Omron Sysmac Studio project 17-408_20171120 (Sysmac Studio 1.19.0.13, StandardProject)

# Controller FS_17_408: NX1P2-9024DT version 1.13
Units and slaves: 節點1 : ASDA-A2-E CoE Drive (E001); 節點2 : ASDA-A2-E CoE Drive (E002)
Axis MC_Axis000, settings changed from default: AxisType=ServoType, FunctionLimit=SingleAxisPTP, UnitsConversion=EnumElement2, UnitsNumerator=1280000, UnitsDenominator=10, WorkGearRatio=16, MaxVelocity=500, MaxJogVelocity=500, HomingMode=BackupAndProximitySignalOn, HomingVelocity=10, HomingApproachVelocity=1, CompensationVelocity=1
Axis MC_Axis001, settings changed from default: AxisNumber=1, AxisType=ServoType, FunctionLimit=SingleAxisPTP, UnitsConversion=EnumElement2, UnitsNumerator=1280000, ReducerUse=EnumElement2, UnitsDenominator=11.75, TravelDistancePerWorkRotation=188, MotorGearRatio=16, MaxVelocity=600, MaxJogVelocity=600, HomingMode=BackupAndProximitySignalOn, HomingVelocity=20, HomingApproachVelocity=1, CompensationVelocity=1
Task PrimaryTask (priority 4, period or condition 2000): prAxis, prMainFlow, prSupplierNFeed, prInit, prError, prConverter

TYPE stAxis : STRUCT
    pbServoOn : BOOL;
    pbReset : BOOL;
    pbSerchHome : BOOL;
    pbJOGForward : BOOL;
    pbJOGBackward : BOOL;
    pbStop : BOOL;
    pbMoveAbs : BOOL;
    bMoveAbsDone : BOOL;
    bHoming : BOOL;
    bServoOn : BOOL;
    bAtPickPosition : BOOL;
    bAtLeavePickPosition : BOOL;
    bAtPutPosition : BOOL;
    bAtTHMoveSavePosition : BOOL;
    lrCurrentPosition : LREAL;
    lrMoveAbsAddData : LREAL;
    lrMoveAbsVelocity : LREAL;
    lrMoveJogVelocity : LREAL;
END_STRUCT END_TYPE

VAR_GLOBAL
    LS_THBack : BOOL;  (* 銅球節流回; at BuiltInIO://cpu/#0/Input_Bit_00; published *)
    LS_THOut : BOOL;  (* 銅球節流出; at BuiltInIO://cpu/#0/Input_Bit_01; published *)
    LS_MoveBack : BOOL;  (* 銅球前後回; at BuiltInIO://cpu/#0/Input_Bit_02; published *)
    LS_MoveOut : BOOL;  (* 銅球前後出; at BuiltInIO://cpu/#0/Input_Bit_03; published *)
    LS_ClipBack : BOOL;  (* 銅球夾持回; at BuiltInIO://cpu/#0/Input_Bit_04; published *)
    LS_ClipOut : BOOL;  (* 銅球夾持出; at BuiltInIO://cpu/#0/Input_Bit_05; published *)
    SNR_MCInPosition : BOOL;  (* 設備定位檢知; at BuiltInIO://cpu/#0/Input_Bit_08; published *)
    SNR_Feed : BOOL;  (* 銅球進料檢知; at BuiltInIO://cpu/#0/Input_Bit_09; published *)
    SNR_Full : BOOL;  (* 銅球滿料檢知; at BuiltInIO://cpu/#0/Input_Bit_10; published *)
    Ex_StartFlag : BOOL;  (* 外部設備送料起動; at BuiltInIO://cpu/#0/Input_Bit_12; published *)
    Ex_ClipOn : BOOL;  (* 外部設備已夾持; at BuiltInIO://cpu/#0/Input_Bit_13; published *)
    SOL_TH : BOOL;  (* 銅球節流電磁閥; at BuiltInIO://cpu/#0/Output_Bit_00; published *)
    SOL_Move : BOOL;  (* 銅球前後電磁閥; at BuiltInIO://cpu/#0/Output_Bit_01; published *)
    SOL_Clip : BOOL;  (* 銅球夾持電磁閥; at BuiltInIO://cpu/#0/Output_Bit_02; published *)
    SOL_FixBack : BOOL;  (* 定位氣壓夾爪回電磁閥; at BuiltInIO://cpu/#0/Output_Bit_03; published *)
    SOL_FixUpBack : BOOL;  (* 上振動定位氣壓夾爪回電磁閥; at BuiltInIO://cpu/#0/Output_Bit_04; published *)
    RY_Full : BOOL;  (* 振動筒繼電器; at BuiltInIO://cpu/#0/Output_Bit_05; published *)
    RY_Feed : BOOL;  (* 平送繼電器; at BuiltInIO://cpu/#0/Output_Bit_06; published *)
    RY_Brake : BOOL;  (* 上下軸剎車繼電器; at BuiltInIO://cpu/#0/Output_Bit_07; published *)
    Ex_FinishFlag : BOOL;  (* 外部設備送料完成; at BuiltInIO://cpu/#0/Output_Bit_08; published *)
    Ex_MachineReday : BOOL;  (* 外部設備可動作; at BuiltInIO://cpu/#0/Output_Bit_09; published *)
    SOL_FixOut : BOOL;  (* 定位氣壓夾爪出電磁閥; at IOBus://unit#2/Output Bit 16 bits/Output Bit 00; published *)
    SOL_FixUpOut : BOOL;  (* 上振動定位氣壓夾爪出電磁閥; at IOBus://unit#2/Output Bit 16 bits/Output Bit 02; published *)
    SOL_FixDownBack : BOOL;  (* 下振動定位氣壓夾爪回電磁閥; at IOBus://unit#2/Output Bit 16 bits/Output Bit 04; published *)
    SOL_FixDownOut : BOOL;  (* 下振動定位氣壓夾爪出電磁閥; at IOBus://unit#2/Output Bit 16 bits/Output Bit 06; published *)
    BZ : BOOL;  (* 蜂鳴器; at IOBus://unit#2/Output Bit 16 bits/Output Bit 01 *)
    YL : BOOL;  (* 黃燈; at IOBus://unit#2/Output Bit 16 bits/Output Bit 03 *)
    GL : BOOL;  (* 綠燈; at IOBus://unit#2/Output Bit 16 bits/Output Bit 05 *)
    RL : BOOL;  (* 紅燈; at IOBus://unit#2/Output Bit 16 bits/Output Bit 07 *)
END_VAR
VAR_GLOBAL CONSTANT
    MC_Axis000 : _sAXIS_REF;  (* at MC://_MC_AX[0] *)
    MC_Axis001 : _sAXIS_REF;  (* at MC://_MC_AX[1] *)
END_VAR
VAR_GLOBAL
    AxUpDown : stAxis;
    AxMove : stAxis;
    CurrentPosition_X : REAL;  (* published *)
    CurrentPosition_Y : REAL;  (* published *)
END_VAR
VAR_GLOBAL RETAIN
    PickPosition_X : REAL;
    PickPosition_Y : REAL;  (* published *)
    LeavePickPosition_X : REAL;  (* published *)
    LeavePickPosition_Y : REAL;  (* published *)
    PutPosition_X : REAL;  (* published *)
    PutPosition_Y : REAL;  (* published *)
END_VAR
VAR_GLOBAL
    SystemReadyStatus : BOOL;  (* published *)
    ErrorStatusTH : BOOL;  (* published *)
    ErrorStatus : BOOL;  (* published *)
    FeedStart : BOOL;  (* published *)
    FeedFinish : BOOL;  (* published *)
    Manual2AutoFlag : BOOL;  (* published *)
    AutoStatus : BOOL;  (* 自動狀態; published *)
    PB_Brake : BOOL;  (* 上下軸剎車; published *)
    PB_TH : BOOL;  (* 節流; published *)
    PB_Move : BOOL;  (* 前後; published *)
    PB_Clip : BOOL;  (* 夾持; published *)
    PB_FixBack : BOOL;  (* 夾爪回; published *)
    PB_FixOut : BOOL;  (* 夾爪出; published *)
    PB_ServoMoveIn : BOOL;  (* 伺服移入; published *)
    PB_ServoMoveOut : BOOL;  (* 伺服移出; published *)
    PB_ServoUp : BOOL;  (* 伺服移上; published *)
    PB_ServoDown : BOOL;  (* 伺服移下; published *)
    PB_SetPickPositionAdd : BOOL;  (* 設定取銅球位置; published *)
    PB_SetLeavePickPositionAdd : BOOL;  (* 設定離開取銅球位置; published *)
    PB_SetPutPositionAdd : BOOL;  (* 設定放銅球位置; published *)
    PB_PickPositionGo : BOOL;  (* 移動至取銅球位置; published *)
    PB_LeavePickPositionGo : BOOL;  (* 移動至離開取銅球位置; published *)
    PB_PutPositionGo : BOOL;  (* 移動至放銅球位置; published *)
    PB_Reset : BOOL;  (* ResetPB; published *)
    PB_ServoOn_Move : BOOL;  (* published *)
    PB_ServoOn_UpDown : BOOL;  (* published *)
    PB_AutoTest : BOOL;  (* published *)
    PB_MachineRun : BOOL;  (* published *)
    PB_LeavePutPositionGo : BOOL;  (* published *)
    State_HomeSerching_Move : BOOL;  (* published *)
    State_Homed_Move : BOOL;  (* published *)
    State_HomeSerching_Updown : BOOL;  (* published *)
    State_Homed_Updown : BOOL;  (* published *)
    State_Homed_MC : BOOL;  (* published *)
    State_Homing_MC : BOOL;  (* published *)
END_VAR
VAR_GLOBAL RETAIN
    SV_ServoMoveJogSpeed : LREAL;  (* 伺服橫移JOG速度; published *)
    SV_ServoMoveJogSpeed_R : REAL;  (* 伺服橫移JOG速度; published *)
    SV_ServoUpdownJogSpeed : LREAL;  (* 伺服上下JOG速度; published *)
    SV_ServoUpdownJogSpeed_R : REAL;  (* 伺服上下JOG速度; published *)
    FullNotExistTime : LINT;  (* published *)
    FullNotExistTime_INT : INT;  (* published *)
    FullExistTime : LINT;  (* published *)
    FullExistTime_INT : INT;  (* published *)
    FullNotExistErrorTime : LINT;  (* published *)
    FullNotExistErrorTime_INT : INT;  (* published *)
    SV_MoveAbsSpeed : LREAL;  (* 伺服橫移ABS速度; published *)
    SV_MoveAbsSpeed_R : REAL;  (* 伺服橫移ABS速度; published *)
    SV_UpDownAbsSpeed : LREAL;  (* 伺服上下ABS速度; published *)
    SV_UpDownAbsSpeed_R : REAL;  (* 伺服上下ABS速度; published *)
    FeedNotExistTime : LINT;  (* published *)
    FeedNotExistTime_INT : INT;  (* published *)
    FeedExistTime : LINT;  (* published *)
    FeedExistTime_INT : INT;  (* published *)
    MachineCount : LINT;  (* published *)
END_VAR
VAR_GLOBAL
    Error_LS_THBack : BOOL;  (* published *)
    Error_LS_THOut : BOOL;  (* published *)
    Error_LS_MoveBack : BOOL;  (* published *)
    Error_LS_MoveOut : BOOL;  (* published *)
    Error_LS_ClipBack : BOOL;  (* published *)
    Error_LS_ClipOut : BOOL;  (* published *)
    Error_SNR_MCInPosition : BOOL;  (* published *)
    Error_SNR_Feed : BOOL;  (* published *)
    Error_SNR_Full : BOOL;  (* published *)
    Error_EStopPB : BOOL;  (* published *)
    Error_Servo_UpDown : BOOL;  (* published *)
    Error_Servo_Move : BOOL;  (* published *)
END_VAR
VAR_GLOBAL RETAIN
    mem_Ex_MachineReady : BOOL;  (* published *)
END_VAR
VAR_GLOBAL
    EStopPB : BOOL;  (* 緊急停止; at BuiltInIO://cpu/#0/Input_Bit_07; published *)
END_VAR

PROGRAM prAxis
VAR
    MC_Power_Ax1 : MC_Power;
    MC_Power_Ax2 : MC_Power;
    MC_Home_Ax1 : MC_Home;
    MC_Home_Ax2 : MC_Home;
    MC_MoveJog_Ax1 : MC_MoveJog;
    MC_MoveJog_Ax2 : MC_MoveJog;
    MC_Reset_Ax1 : MC_Reset;
    MC_Reset_Ax2 : MC_Reset;
    MC_MoveAbsolute_Ax1 : MC_MoveAbsolute;
    MC_MoveAbsolute_Ax2 : MC_MoveAbsolute;
    MC_Stop_Ax1 : MC_Stop;
    MC_Stop_Ax2 : MC_Stop;
END_VAR
VAR_EXTERNAL CONSTANT
    MC_Axis001 : _sAXIS_REF;
END_VAR
VAR_EXTERNAL
    AxMove : stAxis;
END_VAR
VAR_EXTERNAL CONSTANT
    MC_Axis000 : _sAXIS_REF;
END_VAR
VAR_EXTERNAL
    RY_Brake : BOOL;
    PB_Brake : BOOL;
    AxUpDown : stAxis;
    EStopPB : BOOL;
    Error_EStopPB : BOOL;
    PB_Reset : BOOL;
    PB_ServoOn_UpDown : BOOL;
    PB_ServoOn_Move : BOOL;
    PickPosition_Y : REAL;
    PickPosition_X : REAL;
    LeavePickPosition_Y : REAL;
    LeavePickPosition_X : REAL;
    PutPosition_Y : REAL;
    PutPosition_X : REAL;
END_VAR
(*上下軸*)
//Servo on
AxUpDown.pbServoOn:=PB_ServoOn_UpDown;
MC_Power_Ax1(Axis:=MC_Axis000, Enable:=AxUpDown.pbServoOn AND NOT(Error_EStopPB));
//剎車
RY_Brake:=MC_Axis000.DrvStatus.ServoOn OR PB_Brake;
//Reset
MC_Reset_Ax1(Axis:=MC_Axis000, Execute:=AxUpDown.pbReset);
//Home
MC_Home_Ax1(Axis:=MC_Axis000, Execute:=AxUpDown.pbSerchHome AND AxUpDown.bServoOn);
//STOP
MC_Stop_Ax1(Axis:=MC_Axis000, Execute:=AxUpDown.pbStop OR NOT(EStopPB));
//JOG
MC_MoveJog_Ax1(Axis:=MC_Axis000, PositiveEnable:=AxUpDown.pbJOGBackward, NegativeEnable:=AxUpDown.pbJOGForward,
			   Velocity:=AxUpDown.lrMoveJogVelocity,acceleration:=5000,deceleration:=5000);
//絕對定位
MC_MoveAbsolute_Ax1(Axis:=MC_Axis000, Execute:=AxUpDown.pbMoveAbs AND AxUpDown.bServoOn AND MC_Axis000.Details.Homed,
					Position:=AxUpDown.lrMoveAbsAddData,	Velocity:=AxUpDown.lrMoveAbsVelocity,acceleration:=5000,deceleration:=5000,
					Done=>AxUpDown.bMoveAbsDone);

//定義
//Servo On
AxUpDown.bServoOn:=MC_Axis000.DrvStatus.ServoOn;
//找HOME
AxUpDown.bHoming:=MC_Axis000.Status.Homing;
//現在位置
AxUpDown.lrCurrentPosition:=MC_Axis000.Act.Pos;


(*橫移軸*)
//Servo on
AxMove.pbServoOn:=PB_ServoOn_Move;
MC_Power_Ax2(Axis:=MC_Axis001, Enable:=AxMove.pbServoOn AND NOT(Error_EStopPB));
//Reset
MC_Reset_Ax2(Axis:=MC_Axis001, Execute:=AxMove.pbReset);
//Home
MC_Home_Ax2(Axis:=MC_Axis001, Execute:=AxMove.pbSerchHome AND AxMove.bServoOn);
//STOP
MC_Stop_Ax2(Axis:=MC_Axis001, Execute:=AxMove.pbStop OR NOT(EStopPB));
//JOG
MC_MoveJog_Ax2(Axis:=MC_Axis001, PositiveEnable:=AxMove.pbJOGForward, NegativeEnable:=AxMove.pbJOGBackward, Velocity:=AxMove.lrMoveJogVelocity,acceleration:=5000,deceleration:=5000);
//絕對定位
MC_MoveAbsolute_Ax2(Axis:=MC_Axis001, Execute:=AxMove.pbMoveAbs AND AxMove.bServoOn AND MC_Axis001.Details.Homed,
					Position:=AxMove.lrMoveAbsAddData,	Velocity:=AxMove.lrMoveAbsVelocity,acceleration:=5000,deceleration:=5000,
					Done=>AxMove.bMoveAbsDone);

//定義
//Servo On
AxMove.bServoOn:=MC_Axis001.DrvStatus.ServoOn;
//找HOME
AxMove.bHoming:=MC_Axis001.Status.Homing;
//現在位置
AxMove.lrCurrentPosition:=MC_Axis001.Act.Pos;

//伺服位置定義
//取銅球位置
AxUpDown.bAtPickPosition:=(PickPosition_Y-0.01<=AxUpDown.lrCurrentPosition) AND (AxUpDown.lrCurrentPosition<=PickPosition_Y+0.01);
AxMove.bAtPickPosition:=(PickPosition_X-0.01<=AxMove.lrCurrentPosition) AND (AxMove.lrCurrentPosition<=PickPosition_X+0.01);
//離開取銅球位置
AxUpDown.bAtLeavePickPosition:=(LeavePickPosition_Y-0.01<=AxUpDown.lrCurrentPosition) AND (AxUpDown.lrCurrentPosition<=LeavePickPosition_Y+0.01);
AxMove.bAtLeavePickPosition:=(LeavePickPosition_X-0.01<=AxMove.lrCurrentPosition) AND (AxMove.lrCurrentPosition<=LeavePickPosition_X+0.01);
//放銅球位置
AxUpDown.bAtPutPosition:=(PutPosition_Y-0.01<=AxUpDown.lrCurrentPosition) AND (AxUpDown.lrCurrentPosition<=PutPosition_Y+0.01);
AxMove.bAtPutPosition:=(PutPosition_X-0.01<=AxMove.lrCurrentPosition) AND (AxMove.lrCurrentPosition<=PutPosition_X+0.01);

//RESET
AxMove.pbReset:=PB_Reset;
AxUpDown.pbReset:=PB_Reset;
END_PROGRAM

PROGRAM prMainFlow
VAR
    AutoFlow : INT;
    InitFlow : INT;
    F_TRIG1 : F_TRIG;
    R_TRIG_1 : R_TRIG;
    R_TRIG_2 : R_TRIG;
    R_TRIG_3 : R_TRIG;
    R_TRIG_4 : R_TRIG;
    R_TRIG_5 : R_TRIG;
    R_TRIG_6 : R_TRIG;
    R_TRIG_7 : R_TRIG;
    interlockmoveout : BOOL;
    interlockclipout : BOOL;
    interlockFixOut : BOOL;
    interlockmoveback : BOOL;
    interlockclipback : BOOL;
    interlockFixBack : BOOL;
    moveStatus : BOOL;
    clipStatus : BOOL;
    testbit0 : BOOL;
    TON_1 : TON;
    TON_2 : TON;
    TON_3 : TON;
    MC_MoveAbsolute_59 : MC_MoveAbsolute;
    MC_MoveAbsolute_32 : MC_MoveAbsolute;
    MC_MoveAbsolute_62_X : MC_MoveAbsolute;
    MC_MoveAbsolute_62_Y : MC_MoveAbsolute;
    MC_MoveAbsolute_23_X : MC_MoveAbsolute;
    MC_MoveAbsolute_23_Y : MC_MoveAbsolute;
    MC_MoveAbsolute_28_X : MC_MoveAbsolute;
    MC_MoveAbsolute_28_Y : MC_MoveAbsolute;
    MC_MoveAbsolute_53_X : MC_MoveAbsolute;
    MC_MoveAbsolute_53_Y : MC_MoveAbsolute;
    MC_MoveAbsolute_70_X : MC_MoveAbsolute;
    MC_MoveAbsolute_init_X : MC_MoveAbsolute;
    MC_MoveAbsolute_init_Y : MC_MoveAbsolute;
    TON_4 : TON;
    TON_5 : TON;
END_VAR
VAR_EXTERNAL
    SystemReadyStatus : BOOL;
    AutoStatus : BOOL;
    LS_ClipBack : BOOL;
    Ex_StartFlag : BOOL;
    PB_Move : BOOL;
    SOL_Move : BOOL;
    PB_Clip : BOOL;
    SOL_Clip : BOOL;
    AxMove : stAxis;
    PB_ServoMoveOut : BOOL;
    PB_ServoMoveIn : BOOL;
    AxUpDown : stAxis;
    PB_ServoUp : BOOL;
    PB_ServoDown : BOOL;
END_VAR
VAR_EXTERNAL CONSTANT
    MC_Axis001 : _sAXIS_REF;
    MC_Axis000 : _sAXIS_REF;
END_VAR
VAR_EXTERNAL
    SV_ServoUpdownJogSpeed : LREAL;
    SV_ServoMoveJogSpeed : LREAL;
    PB_SetPickPositionAdd : BOOL;
    PB_SetLeavePickPositionAdd : BOOL;
    PB_SetPutPositionAdd : BOOL;
    PB_PickPositionGo : BOOL;
    PB_LeavePickPositionGo : BOOL;
    PB_PutPositionGo : BOOL;
    LS_MoveBack : BOOL;
    SV_UpDownAbsSpeed : LREAL;
    SV_MoveAbsSpeed : LREAL;
    LS_MoveOut : BOOL;
    LS_ClipOut : BOOL;
    EStopPB : BOOL;
    Error_EStopPB : BOOL;
    ErrorStatus : BOOL;
    RY_Brake : BOOL;
    FeedStart : BOOL;
    FeedFinish : BOOL;
    LS_THBack : BOOL;
    SOL_TH : BOOL;
    Manual2AutoFlag : BOOL;
    MachineCount : LINT;
    PB_FixBack : BOOL;
    SOL_FixBack : BOOL;
    SOL_FixUpBack : BOOL;
    SOL_FixDownBack : BOOL;
    SOL_FixOut : BOOL;
    SOL_FixUpOut : BOOL;
    SOL_FixDownOut : BOOL;
    PB_FixOut : BOOL;
    PB_AutoTest : BOOL;
    Ex_FinishFlag : BOOL;
    PB_MachineRun : BOOL;
    Ex_ClipOn : BOOL;
    Ex_MachineReday : BOOL;
    mem_Ex_MachineReady : BOOL;
    PB_LeavePutPositionGo : BOOL;
    LeavePickPosition_X : REAL;
    LeavePickPosition_Y : REAL;
    PickPosition_X : REAL;
    PickPosition_Y : REAL;
    PutPosition_X : REAL;
    PutPosition_Y : REAL;
    CurrentPosition_X : REAL;
    CurrentPosition_Y : REAL;
END_VAR
(*************************************************************************
程序名稱:主要取放流程
作者:蔡相偉
版本,日期,版本資訊:
1.0.0	2017/7/10		初始版本
PowerOn=0
Idle=1
	|____________________________
	|											|
無夾取=20							有夾取=50
前後回=21							前後回=51
伺服移至離開取料點=61		伺服移至放料離開點點=31
伺服起動=62						伺服起動=32
伺服到位=63						伺服到位=33
伺服移至取料點=22			伺服移至放料點=52
伺服起動=23						伺服起動=53
伺服到位=24						伺服到位=54
前後出=25							前後出=55
											放料完成=80
夾取出=26							夾取回=56
伺服至離開取料點=27			前後回=57
伺服起動=28						伺服移至放料離開點點=58
伺服到位=29						伺服起動=59
前後回=30							伺服到位=60
											伺服移至取料離開點=70
											伺服到位=71
*************************************************************************)
IF NOT(AutoStatus) OR ErrorStatus THEN
	PB_MachineRun:=FALSE;
END_IF;

//PowerOn=0
IF not(SystemReadyStatus) OR NOT(AutoStatus) OR ErrorStatus OR Error_EStopPB THEN
	AutoFlow:=0;
	Ex_FinishFlag:=FALSE;
END_IF;
//Idle=1
IF AutoFlow=0 AND SystemReadyStatus AND AutoStatus AND NOT(Error_EStopPB) AND NOT(ErrorStatus) THEN
	AutoFlow:=1;
END_IF;
IF AutoFlow=71 THEN
	AutoFlow:=1;
END_IF;

//無夾取=20
testbit0:=PB_AutoTest;
IF AutoFlow=1 AND LS_ClipBack AND NOT(LS_ClipOut) AND NOT(SOL_Clip) AND PB_MachineRun THEN
	AutoFlow:=20;
END_IF;

//前後回=21
IF AutoFlow=20 THEN
	AutoFlow:=21;
END_IF;
(*IF AutoFlow=57 AND LS_MoveBack AND NOT(LS_MoveOut) AND NOT(SOL_Move) AND (Ex_StartFlag OR testbit0) THEN
	AutoFlow:=22;
END_IF;*)
//伺服至離開取料點=61
IF AutoFlow=21 AND LS_MoveBack AND NOT(LS_MoveOut) AND NOT(SOL_Move) THEN
	AutoFlow:=61;
END_IF;

//伺服起動=62
IF AutoFlow=61 THEN
	AutoFlow:=62;
END_IF;
MC_MoveAbsolute_62_X(Axis:=MC_Axis001, Execute:=AutoFlow=62  AND AxMove.bServoOn AND MC_Axis001.Details.Homed,
					Position:=LeavePickPosition_X,	Velocity:=SV_MoveAbsSpeed,acceleration:=5000,deceleration:=5000);
MC_MoveAbsolute_62_Y(Axis:=MC_Axis000, Execute:=AutoFlow=62  AND AxUpDown.bServoOn AND MC_Axis000.Details.Homed,
					Position:=LeavePickPosition_Y,	Velocity:=SV_UpDownAbsSpeed,acceleration:=5000,deceleration:=5000);

//伺服到位=63
IF AutoFlow=62 AND MC_MoveAbsolute_62_X.Done AND MC_MoveAbsolute_62_Y.Done THEN
	AutoFlow:=63;
END_IF;

//伺服移至取料點=22
IF AutoFlow=63 THEN
	AutoFlow:=22;
END_IF;

//伺服起動=23
IF AutoFlow=22 THEN
	AutoFlow:=23;
END_IF;
MC_MoveAbsolute_23_X(Axis:=MC_Axis001, Execute:=AutoFlow=23 AND AxMove.bServoOn AND MC_Axis001.Details.Homed,
					Position:=PickPosition_X,	Velocity:=SV_MoveAbsSpeed,acceleration:=5000,deceleration:=5000);
MC_MoveAbsolute_23_Y(Axis:=MC_Axis000, Execute:=AutoFlow=23 AND AxUpDown.bServoOn AND MC_Axis000.Details.Homed,
					Position:=PickPosition_Y,	Velocity:=SV_UpDownAbsSpeed,acceleration:=5000,deceleration:=5000);
//伺服到位=24
IF AutoFlow=23 AND MC_MoveAbsolute_23_X.Done AND MC_MoveAbsolute_23_Y.Done THEN
	AutoFlow:=24;
END_IF;

//前後出=25
IF AutoFlow=24 AND NOT(AxMove.pbMoveAbs) AND NOT(AxUpDown.pbMoveAbs) AND LS_THBack AND NOT(SOL_TH) THEN
	AutoFlow:=25;
END_IF;

//夾取出=26
IF AutoFlow=25 AND LS_MoveOut THEN
	AutoFlow:=26;
END_IF;

//伺服至離開取料點=27
IF AutoFlow=26 AND LS_ClipOut AND NOT(LS_ClipBack) AND (SOL_Clip) THEN
	AutoFlow:=27;
END_IF;

//伺服起動=28
IF AutoFlow=27 THEN
	AutoFlow:=28;
END_IF;
MC_MoveAbsolute_28_X(Axis:=MC_Axis001, Execute:=AutoFlow=28 AND AxMove.bServoOn AND MC_Axis001.Details.Homed,
					Position:=LeavePickPosition_X,	Velocity:=SV_MoveAbsSpeed,acceleration:=5000,deceleration:=5000);
MC_MoveAbsolute_28_Y(Axis:=MC_Axis000, Execute:=AutoFlow=28 AND AxUpDown.bServoOn AND MC_Axis000.Details.Homed,
					Position:=LeavePickPosition_Y,	Velocity:=SV_UpDownAbsSpeed,acceleration:=5000,deceleration:=5000);
//伺服到位=29
IF AutoFlow=28 AND MC_MoveAbsolute_28_X.Done AND MC_MoveAbsolute_28_Y.Done THEN
	AutoFlow:=29;
END_IF;
IF AutoFlow=29 THEN
	FeedStart:=TRUE;
END_IF;
IF FeedFinish OR AutoFlow=0 THEN
	FeedStart:=FALSE;
END_IF;

//前後回=30
IF AutoFlow=29 THEN
	AutoFlow:=30;
END_IF;

//********************************************************************************************************
//有夾取=50
IF AutoFlow=1 AND (LS_ClipOut) AND NOT(LS_ClipBack) AND SOL_Clip THEN
	AutoFlow:=50;
END_IF;

//前後回=51
IF AutoFlow=50 THEN
	AutoFlow:=51;
END_IF;
//伺服移至放料離開點點=31
IF AutoFlow=30 AND LS_MoveBack AND (Ex_StartFlag OR testbit0) THEN
	AutoFlow:=31;
END_IF;
IF AutoFlow=51 AND LS_MoveBack AND (Ex_StartFlag OR testbit0) THEN
	AutoFlow:=31;
	
END_IF;

//伺服起動=32
IF  AutoFlow=31 THEN
	AutoFlow:=32;
END_IF;
MC_MoveAbsolute_32(Axis:=MC_Axis001, Execute:=AutoFlow=32 AND AxMove.bServoOn AND MC_Axis001.Details.Homed,
					Position:=PutPosition_X,	Velocity:=SV_MoveAbsSpeed,acceleration:=5000,deceleration:=5000);
//伺服到位=33
IF AutoFlow=32 AND MC_MoveAbsolute_32.Done THEN
	AutoFlow:=33;
END_IF;

//伺服移至放料點=52
IF AutoFlow=33 THEN
	AutoFlow:=52;
END_IF;

//伺服起動=53
IF AutoFlow=52 THEN
	AutoFlow:=53;
END_IF;
MC_MoveAbsolute_53_X(Axis:=MC_Axis001, Execute:=AutoFlow=53 AND AxMove.bServoOn AND MC_Axis001.Details.Homed,
					Position:=PutPosition_X,	Velocity:=SV_MoveAbsSpeed,acceleration:=5000,deceleration:=5000);
MC_MoveAbsolute_53_Y(Axis:=MC_Axis000, Execute:=AutoFlow=53 AND AxUpDown.bServoOn AND MC_Axis000.Details.Homed,
					Position:=PutPosition_Y,	Velocity:=SV_UpDownAbsSpeed,acceleration:=5000,deceleration:=5000);
//伺服到位=54
IF AutoFlow=53 AND MC_MoveAbsolute_53_X.Done AND MC_MoveAbsolute_53_Y.Done THEN
	AutoFlow:=54;
	mem_Ex_MachineReady:=FALSE;
END_IF;

//前後出=55
IF AutoFlow=54 AND NOT(mem_Ex_MachineReady) THEN
	AutoFlow:=55;
END_IF;
//放料完成=80
TON_5(In:=AutoFlow=55 AND LS_MoveOut, PT:=t#500ms);
IF AutoFlow=55 AND TON_5.Q THEN
	AutoFlow:=80;
END_IF;
IF AutoFlow=80 THEN
	Ex_FinishFlag:=TRUE;
END_IF;

//夾取回=56
TON_4(In:=AutoFlow=80  AND Ex_ClipOn, PT:=t#500ms);
IF AutoFlow=80 AND TON_4.Q THEN
	AutoFlow:=56;
	MachineCount:=MachineCount+1;
END_IF;

//前後回=57
IF AutoFlow=56 AND LS_ClipBack THEN
	AutoFlow:=57;
END_IF;
Ex_MachineReday:=mem_Ex_MachineReady;
//伺服移至離開放料點=58
IF AutoFlow=57 AND LS_MoveBack AND NOT(LS_MoveOut) AND NOT(SOL_Move) AND NOT(Ex_StartFlag) AND NOT(testbit0) THEN
	AutoFlow:=58;
	mem_Ex_MachineReady:=TRUE;
	Ex_FinishFlag:=FALSE;
END_IF;

//伺服起動=59
IF AutoFlow=58 THEN
	AutoFlow:=59;
END_IF;
MC_MoveAbsolute_59(Axis:=MC_Axis000, Execute:=AutoFlow=59 AND AxUpDown.bServoOn AND MC_Axis000.Details.Homed,
					Position:=LeavePickPosition_Y,	Velocity:=SV_UpDownAbsSpeed,acceleration:=5000,deceleration:=5000);
//伺服到位=60
IF AutoFlow=59 AND MC_MoveAbsolute_59.Done  THEN
	AutoFlow:=60;
END_IF;

//伺服移至取料離開點=70
IF AutoFlow=60 THEN
	AutoFlow:=70;
END_IF;
MC_MoveAbsolute_70_X(Axis:=MC_Axis001, Execute:=AutoFlow=70 AND AxMove.bServoOn AND MC_Axis001.Details.Homed,
					Position:=PickPosition_X,	Velocity:=SV_MoveAbsSpeed,acceleration:=5000,deceleration:=5000);
//伺服到位=71
IF AutoFlow=70 AND MC_MoveAbsolute_70_X.Done  THEN
	AutoFlow:=71;
END_IF;

//***************************************************************************************************
//TON_1(In:=AutoFlow=23 OR AutoFlow=28 OR AutoFlow=53 (*OR AutoFlow=59*) OR AutoFlow=62 OR InitFlow=5, PT:=t#100ms);
//R_TRIG_6(Clk:=AutoFlow=23 OR AutoFlow=28 OR AutoFlow=53 (*OR AutoFlow=59*) OR AutoFlow=62 OR InitFlow=5);
//IF R_TRIG_6.Q THEN
//	AxMove.pbMoveAbs:=TRUE;
//	AxUpDown.pbMoveAbs:=TRUE;
//END_IF;
//***************************************************************************************************
//異常
IF NOT(EStopPB) OR ErrorStatus THEN
	AutoFlow:=0;
	SOL_Clip:=FALSE;
END_IF;

//***************************************************************************************************
(*手動*)
(*前後電磁閥*)
R_TRIG_1(CLK:=PB_Move AND NOT(AutoStatus));
interlockmoveback:=TRUE;
interlockmoveout:=(AxUpDown.bAtPickPosition AND AxMove.bAtPickPosition) OR (AxUpDown.bAtPutPosition AND AxMove.bAtPutPosition);
(*SET*)
IF ((R_TRIG_1.Q AND NOT(moveStatus)) OR AutoFlow=25 OR AutoFlow=55) AND interlockmoveout THEN
	SOL_Move:=TRUE;
END_IF;
(*RESET*)
IF ((R_TRIG_1.Q AND (moveStatus)) OR AutoFlow=21 OR AutoFlow=30 OR AutoFlow=51 OR AutoFlow=57 OR InitFlow=3) AND interlockmoveback THEN
	SOL_Move:=FALSE;
END_IF;
(*STATUS*)
moveStatus:=SOL_Move;

(*夾持電磁閥*)
R_TRIG_2(CLK:=PB_Clip AND NOT(AutoStatus));
interlockclipback:=TRUE;
interlockclipout:=TRUE;
(*SET*)
IF ((R_TRIG_2.Q AND NOT(clipStatus)) OR AutoFlow=26) AND interlockclipout THEN
	SOL_Clip:=TRUE;
END_IF;
(*RESET*)
IF ((R_TRIG_2.Q AND (clipStatus)) OR AutoFlow=56 OR InitFlow=2) AND interlockclipback THEN
	SOL_Clip:=FALSE;
END_IF;
(*STATUS*)
clipStatus:=SOL_Clip;

(*伺服移下*)
AxUpDown.pbJOGForward:=AxUpDown.bServoOn and PB_ServoDown AND NOT(AutoStatus);

(*伺服移上*)
AxUpDown.pbJOGBackward:=AxUpDown.bServoOn and PB_ServoUp AND NOT(AutoStatus);

(*伺服移回*)
AxMove.pbJOGForward:=AxMove.bServoOn and PB_ServoMoveOut AND NOT(AutoStatus);

(*伺服移出*)
AxMove.pbJOGBackward:=AxMove.bServoOn and PB_ServoMoveIn AND NOT(AutoStatus);

(*JOG速度*)
AxUpDown.lrMoveJogVelocity:=SV_ServoUpdownJogSpeed;
AxMove.lrMoveJogVelocity:=SV_ServoMoveJogSpeed;

//***************************************************************************************************
(*設定位置*)
//取銅球位置
IF PB_SetPickPositionAdd AND NOT(AutoStatus) THEN
	PickPosition_Y:=LREAL_TO_REAL(AxUpDown.lrCurrentPosition);
	PickPosition_X:=LREAL_TO_REAL(AxMove.lrCurrentPosition);
END_IF;
//離開取銅球位置
IF PB_SetLeavePickPositionAdd AND NOT(AutoStatus) THEN
	LeavePickPosition_Y:=LREAL_TO_REAL(AxUpDown.lrCurrentPosition);
	LeavePickPosition_X:=LREAL_TO_REAL(AxMove.lrCurrentPosition);
END_IF;
//放銅球位置
IF PB_SetPutPositionAdd AND NOT(AutoStatus) THEN
	PutPosition_Y:=LREAL_TO_REAL(AxUpDown.lrCurrentPosition);
	PutPosition_X:=LREAL_TO_REAL(AxMove.lrCurrentPosition);
END_IF;
//當前位置
CurrentPosition_X:=LREAL_TO_REAL(AxMove.lrCurrentPosition);
CurrentPosition_Y:=LREAL_TO_REAL(AxUpDown.lrCurrentPosition);
(*************************************************************************
程序名稱:RESET流程
作者:蔡相偉
版本,日期,版本資訊:
1.0.0	2017/7/14		初始版本
PowerOn=0
Idle=1
夾爪回=2
前後回=3
伺服移至0點=4
伺服起動=5
伺服到位=6
*************************************************************************)
//PowerOn=0
IF NOT(SystemReadyStatus) THEN
	InitFlow:=0;
END_IF;
//Idle=1
IF InitFlow=0 AND SystemReadyStatus THEN
	InitFlow:=1;
END_IF;
IF InitFlow=7 THEN
	InitFlow:=1;
END_IF;

//夾爪回=2
F_TRIG1(Clk:=ErrorStatus);
IF InitFlow=1 AND F_TRIG1.Q THEN
	InitFlow:=2;
END_IF;

//前後回=3
IF InitFlow=2 AND LS_ClipBack THEN
	InitFlow:=3;
END_IF;

//伺服移離開取銅球點=4
TON_2(In:=InitFlow=3 AND LS_MoveBack AND RY_Brake, PT:=t#1s);
IF InitFlow=3 AND TON_2.Q THEN
	InitFlow:=4;
END_IF;
//MC_MoveAbsolute_init_X(Axis:=MC_Axis001, Execute:=InitFlow=4 AND AxMove.bServoOn AND MC_Axis001.Details.Homed,
//					Position:=LeavePickPosition_X,	Velocity:=SV_MoveAbsSpeed,acceleration:=5000,deceleration:=5000);
MC_MoveAbsolute_init_Y(Axis:=MC_Axis000, Execute:=InitFlow=4 AND AxUpDown.bServoOn AND MC_Axis000.Details.Homed,
					Position:=LeavePickPosition_Y,	Velocity:=SV_UpDownAbsSpeed,acceleration:=5000,deceleration:=5000);

//伺服到位=5
IF InitFlow=4 AND MC_MoveAbsolute_init_Y.Done  THEN
	InitFlow:=5;
END_IF;

//伺服go=6
IF InitFlow=5 THEN
	InitFlow:=6;
END_IF;
MC_MoveAbsolute_init_X(Axis:=MC_Axis001, Execute:=InitFlow=6 AND AxMove.bServoOn AND MC_Axis001.Details.Homed,
				Position:=LeavePickPosition_X,	Velocity:=SV_MoveAbsSpeed,acceleration:=5000,deceleration:=5000);
//伺服到位=7
IF InitFlow=6 AND MC_MoveAbsolute_init_X.Done THEN
	InitFlow:=7;
END_IF;

//***************************************************************************************************
(*定位控制*)
//取銅球位置
R_TRIG_3(Clk:=PB_PickPositionGo AND NOT(AutoStatus) AND AxMove.bServoOn AND AxUpDown.bServoOn AND MC_Axis000.Details.Homed AND MC_Axis001.Details.Homed AND LS_MoveBack AND NOT(SOL_Move));
IF R_TRIG_3.Q THEN
	AxUpDown.lrMoveAbsAddData:=PickPosition_Y;
	AxMove.lrMoveAbsAddData:=PickPosition_X;
	AxUpDown.lrMoveAbsVelocity:=SV_UpDownAbsSpeed;
	AxMove.lrMoveAbsVelocity:=SV_MoveAbsSpeed;
	IF (AxUpDown.lrMoveAbsAddData=PickPosition_Y) AND (AxMove.lrMoveAbsAddData=PickPosition_X) THEN
		AxUpDown.pbMoveAbs:=TRUE;
		AxMove.pbMoveAbs:=TRUE;
	END_IF;
END_IF;

//離開取銅球位置
R_TRIG_4(Clk:=PB_LeavePickPositionGo AND NOT(AutoStatus) AND AxMove.bServoOn AND AxUpDown.bServoOn AND MC_Axis000.Details.Homed AND MC_Axis001.Details.Homed);
IF R_TRIG_4.Q THEN
	AxUpDown.lrMoveAbsAddData:=LeavePickPosition_Y;
	AxMove.lrMoveAbsAddData:=LeavePickPosition_X;
	AxUpDown.lrMoveAbsVelocity:=SV_UpDownAbsSpeed;
	AxMove.lrMoveAbsVelocity:=SV_MoveAbsSpeed;
	IF (AxUpDown.lrMoveAbsAddData=LeavePickPosition_Y) AND (AxMove.lrMoveAbsAddData=LeavePickPosition_X) THEN
		AxUpDown.pbMoveAbs:=TRUE;
		AxMove.pbMoveAbs:=TRUE;
	END_IF;
END_IF;

//放銅球位置
R_TRIG_5(Clk:=PB_PutPositionGo AND NOT(AutoStatus) AND AxMove.bServoOn AND AxUpDown.bServoOn AND MC_Axis000.Details.Homed AND MC_Axis001.Details.Homed AND LS_MoveBack AND NOT(SOL_Move));
IF R_TRIG_5.Q THEN
	AxUpDown.lrMoveAbsAddData:=PutPosition_Y;
	AxMove.lrMoveAbsAddData:=PutPosition_X;
	AxUpDown.lrMoveAbsVelocity:=SV_UpDownAbsSpeed;
	AxMove.lrMoveAbsVelocity:=SV_MoveAbsSpeed;
	IF (AxUpDown.lrMoveAbsAddData=PutPosition_Y) AND (AxMove.lrMoveAbsAddData=PutPosition_X) THEN
		AxUpDown.pbMoveAbs:=TRUE;
		AxMove.pbMoveAbs:=TRUE;
	END_IF;
END_IF;
//離開放銅球位置
R_TRIG_7(Clk:=PB_LeavePutPositionGo AND NOT(AutoStatus) AND AxMove.bServoOn AND AxUpDown.bServoOn AND MC_Axis000.Details.Homed AND MC_Axis001.Details.Homed AND LS_MoveBack AND NOT(SOL_Move));
IF R_TRIG_7.Q THEN
	AxUpDown.lrMoveAbsAddData:=LeavePickPosition_Y;
	AxMove.lrMoveAbsAddData:=PutPosition_X;
	AxUpDown.lrMoveAbsVelocity:=SV_UpDownAbsSpeed;
	AxMove.lrMoveAbsVelocity:=SV_MoveAbsSpeed;
	IF (AxUpDown.lrMoveAbsAddData=LeavePickPosition_Y) AND (AxMove.lrMoveAbsAddData=PutPosition_X) THEN
		AxUpDown.pbMoveAbs:=TRUE;
		AxMove.pbMoveAbs:=TRUE;
	END_IF;
END_IF;
//到達位置
IF AxUpDown.bMoveAbsDone OR NOT(EStopPB) THEN
	AxUpDown.pbMoveAbs:=FALSE;
END_IF;
IF AxMove.bMoveAbsDone OR NOT(EStopPB) THEN
	AxMove.pbMoveAbs:=FALSE;
END_IF;

//定位氣缸
//移位歸電磁閥
interlockFixBack:=TRUE;
IF (PB_FixBack) AND NOT(AutoStatus) AND interlockMoveBack THEN
	SOL_FixBack:=TRUE;
	SOL_FixUpBack:=TRUE;
	SOL_FixDownBack:=TRUE;
	SOL_FixOut:=FALSE;
	SOL_FixUpOut:=FALSE;
	SOL_FixDownOut:=FALSE;
END_IF;

//移位出電磁閥
interlockFixOut:=TRUE;
IF (PB_FixOut) AND NOT(AutoStatus) AND interlockFixOut THEN
	SOL_FixBack:=FALSE;
	SOL_FixUpBack:=FALSE;
	SOL_FixDownBack:=FALSE;
	SOL_FixOut:=TRUE;
	SOL_FixUpOut:=TRUE;
	SOL_FixDownOut:=TRUE;
END_IF;

TON_3(In:=SOL_FixBack OR SOL_FixOut, PT:=t#1s);
IF TON_3.Q THEN
	SOL_FixBack:=FALSE;
	SOL_FixUpBack:=FALSE;
	SOL_FixDownBack:=FALSE;
	SOL_FixOut:=FALSE;
	SOL_FixUpOut:=FALSE;
	SOL_FixDownOut:=FALSE;
END_IF;
END_PROGRAM

PROGRAM prSupplierNFeed
VAR
    BallSupplier : Full;
    BallFeeder : fbFeed;
END_VAR
VAR_EXTERNAL
    SNR_Full : BOOL;
    FullExistTime : LINT;
    FullNotExistErrorTime : LINT;
    RY_Full : BOOL;
    Error_SNR_Full : BOOL;
    Error_LS_THBack : BOOL;
    Error_LS_THOut : BOOL;
    FeedStart : BOOL;
    SNR_Feed : BOOL;
    PB_Reset : BOOL;
    LS_THBack : BOOL;
    LS_THOut : BOOL;
    PB_TH : BOOL;
    Error_SNR_Feed : BOOL;
    FeedFinish : BOOL;
    RY_Feed : BOOL;
    SOL_TH : BOOL;
    FeedNotExistTime : LINT;
    FeedExistTime : LINT;
    FullNotExistTime : LINT;
END_VAR
BallSupplier();
BallSupplier.bFullSNR:=SNR_Full;
BallSupplier.iItemNotExistDelayTime:=FullNotExistTime;
BallSupplier.iItemExistTime:=FullExistTime;
BallSupplier.iItemNotExistErrorTime:=FullNotExistErrorTime;
RY_Full:=BallSupplier.bFullRY;
Error_SNR_Full:=BallSupplier.bFullSNRError;

BallFeeder();
BallFeeder.bErrorTHBack:=Error_LS_THBack;
BallFeeder.bErrorTHOut:=Error_LS_THOut;
BallFeeder.bFeedStart:=FeedStart;
BallFeeder.bInterlock_thback:=TRUE;
BallFeeder.bInterlock_thout:=TRUE;
BallFeeder.bObjSNR:=SNR_Feed;
BallFeeder.bReset:=PB_Reset;
BallFeeder.bSupplierRY:=RY_Full;
BallFeeder.bTHBackLS:=LS_THBack;
BallFeeder.bTHOutLS:=LS_THOut;
BallFeeder.bTHPB:=PB_TH;
BallFeeder.wNoObjDelayTime:=FeedNotExistTime;
BallFeeder.wObjectExistDelayTime:=FeedExistTime;
Error_SNR_Feed :=BallFeeder.bFeedError;
FeedFinish:= BallFeeder.bFeedFinish;
RY_Feed:= BallFeeder.bFeedRY;
SOL_TH:= BallFeeder.bTHSOL;
END_PROGRAM

PROGRAM prInit
VAR
    SystemInitFlow : INT := 0;
    TON1 : TON;
    TON_3 : TON;
    R_TRIG_3 : R_TRIG;
END_VAR
VAR_EXTERNAL
    AutoStatus : BOOL;
    SystemReadyStatus : BOOL;
END_VAR
VAR_EXTERNAL CONSTANT
    MC_Axis000 : _sAXIS_REF;
    MC_Axis001 : _sAXIS_REF;
END_VAR
VAR_EXTERNAL
    AxMove : stAxis;
    AxUpDown : stAxis;
    SOL_Clip : BOOL;
    LS_ClipBack : BOOL;
    SOL_Move : BOOL;
    LS_MoveBack : BOOL;
    EStopPB : BOOL;
    Error_EStopPB : BOOL;
    RY_Brake : BOOL;
    ErrorStatus : BOOL;
    ErrorStatusTH : BOOL;
    Error_SNR_Full : BOOL;
    Manual2AutoFlag : BOOL;
    BZ : BOOL;
    RL : BOOL;
    GL : BOOL;
    YL : BOOL;
    Error_SNR_Feed : BOOL;
    PB_ServoOn_UpDown : BOOL;
    PB_ServoOn_Move : BOOL;
END_VAR
(******************************************************************
程式:系統初始化
作者:蔡相偉
版本資訊:1.0.0		2016/5/26

全部狀態RESET=0
伺服上電=1
伺服未回HOME=2
伺服Servo on=3
伺服Ready=4
夾爪回=5
夾爪前後回=6
伺服上下軸Serch Home=7
伺服上下軸Serch Home中=8
伺服上下軸Serch Home完成=9
伺服橫移軸Serch Home=10
伺服橫移軸Serch Home中=11
伺服橫移軸Serch Home完成=12
自動SET=13
系統READY SET=14
Init完成=15
******************************************************************)
//全部狀態RESET=0
IF P_First_Run THEN
	SystemInitFlow:=0;
	AutoStatus:=FALSE;
	SystemReadyStatus:=FALSE;
END_IF;

//伺服上電=1
IF SystemInitFlow=0 AND EStopPB AND NOT(Error_EStopPB) AND NOT(AutoStatus) AND NOT(SystemReadyStatus) AND MC_Axis000.DrvStatus.MainPower AND MC_Axis001.DrvStatus.MainPower THEN
	SystemInitFlow:=1;
END_IF;

//伺服未回HOME=2
IF SystemInitFlow=1 AND (NOT(MC_Axis000.Details.Homed) OR NOT(MC_Axis001.Details.Homed)) THEN
	SystemInitFlow:=2;
END_IF;

//伺服Servo on=3
IF SystemInitFlow=2 THEN
	SystemInitFlow:=3;
END_IF;
IF SystemInitFlow=3 THEN
	PB_ServoOn_UpDown:=TRUE;
	PB_ServoOn_Move:=TRUE;
END_IF;

//伺服Ready=4
IF SystemInitFlow=3 AND AxMove.bServoOn AND AxUpDown.bServoOn AND MC_Axis000.DrvStatus.Ready AND MC_Axis001.DrvStatus.Ready THEN
	SystemInitFlow:=4;
END_IF;

//夾爪回=5
TON1(In:=SystemInitFlow=4 AND RY_Brake, PT:=t#1s);
IF SystemInitFlow=4 AND TON1.Q THEN
	SystemInitFlow:=5;
END_IF;
IF SystemInitFlow=5 THEN
	SOL_Clip:=FALSE;
END_IF;

//夾爪前後回=6
IF SystemInitFlow=5 AND LS_ClipBack THEN
	SystemInitFlow:=6;
END_IF;
IF SystemInitFlow=6 THEN
	SOL_Move:=FALSE;
END_IF;

//伺服上下軸Serch Home=7
IF SystemInitFlow=6 AND LS_MoveBack THEN
	SystemInitFlow:=7;
END_IF;
IF SystemInitFlow=7 THEN
	AxUpDown.pbSerchHome:=TRUE;
END_IF;

//伺服上下軸Serch Home中=8
IF SystemInitFlow=7 AND AxUpDown.bHoming THEN
	AxUpDown.pbSerchHome:=FALSE;
	SystemInitFlow:=8;
END_IF;

//伺服上下軸Serch Home完成=9
IF SystemInitFlow=8 AND NOT(AxUpDown.bHoming) THEN
	SystemInitFlow:=9;
END_IF;

//伺服橫移軸Serch Home=10
IF SystemInitFlow=9 AND MC_Axis000.Details.Homed THEN
	SystemInitFlow:=10;
END_IF;
IF SystemInitFlow=10 THEN
	AxMove.pbSerchHome:=TRUE;
END_IF;

//伺服橫移軸Serch Home中=11
IF SystemInitFlow=10 AND AxMove.bHoming THEN
	AxMove.pbSerchHome:=FALSE;
	SystemInitFlow:=11;
END_IF;

//伺服橫移軸Serch Home完成=12
IF SystemInitFlow=11 AND NOT(AxMove.bHoming) THEN
	SystemInitFlow:=12;
END_IF;

//自動SET=13
IF SystemInitFlow=12 AND MC_Axis001.Details.Homed THEN
	SystemInitFlow:=13;
END_IF;
IF SystemInitFlow=13 THEN
	AutoStatus:=TRUE;
END_IF;

//系統READY SET=14
IF SystemInitFlow=13 AND AutoStatus THEN
	SystemInitFlow:=14;
END_IF;
IF SystemInitFlow=14 THEN
	SystemReadyStatus:=TRUE;
END_IF;

//Init完成=15
IF SystemInitFlow=14 AND SystemReadyStatus THEN
	SystemInitFlow:=15;
END_IF;

//******************************************************************
//手動轉自動
R_TRIG_3(CLK:= AutoStatus ,Q=> Manual2AutoFlag );

(******************************************************************
程式:燈號及蜂鳴器
作者:蔡相偉
版本資訊:1.0.0		2016/5/26
******************************************************************)
//BZ停止
TON_3(IN:=ErrorStatus OR ErrorStatusTH OR Error_SNR_Feed , PT:=t#2s);

//BZ
IF (ErrorStatus OR ErrorStatusTH OR Error_SNR_Feed) AND NOT(TON_3.Q) THEN
	BZ:=TRUE;
	ELSE
	BZ:=FALSE;
END_IF;
//紅燈
IF ErrorStatus OR ErrorStatusTH OR Error_SNR_Feed THEN
	RL:=TRUE;
	ELSE
	RL:=FALSE;
END_IF;
//綠燈
IF NOT(ErrorStatus) AND
	NOT(ErrorStatusTH) AND NOT(Error_SNR_Feed) AND NOT(Error_SNR_Full) THEN
	GL:=TRUE;
	ELSE
	GL:=FALSE;
END_IF;
//黃燈
IF Error_SNR_Full THEN
	YL:=TRUE;
	ELSE
	YL:=FALSE;
END_IF;
END_PROGRAM

PROGRAM prError
VAR
    TON1 : array[0..10] of TON;
END_VAR
VAR_EXTERNAL
    PB_Reset : BOOL;
    SOL_TH : BOOL;
    Error_LS_THBack : BOOL;
    LS_THOut : BOOL;
    Error_LS_THOut : BOOL;
    SOL_Move : BOOL;
    LS_MoveBack : BOOL;
    Error_LS_MoveBack : BOOL;
    LS_MoveOut : BOOL;
    Error_LS_MoveOut : BOOL;
    SOL_Clip : BOOL;
    LS_ClipBack : BOOL;
    Error_LS_ClipBack : BOOL;
    LS_ClipOut : BOOL;
    Error_LS_ClipOut : BOOL;
    EStopPB : BOOL;
    Error_EStopPB : BOOL;
    AutoStatus : BOOL;
    LS_THBack : BOOL;
    ErrorStatus : BOOL;
    ErrorStatusTH : BOOL;
END_VAR
VAR_EXTERNAL CONSTANT
    MC_Axis000 : _sAXIS_REF;
END_VAR
VAR_EXTERNAL
    Error_Servo_UpDown : BOOL;
    Error_Servo_Move : BOOL;
END_VAR
VAR_EXTERNAL CONSTANT
    MC_Axis001 : _sAXIS_REF;
END_VAR
VAR_EXTERNAL
    SNR_MCInPosition : BOOL;
    SystemReadyStatus : BOOL;
    Error_SNR_MCInPosition : BOOL;
END_VAR
IF AutoStatus AND NOT(PB_Reset) THEN
	(*節流歸磁簧開關*)
	TON1[0](IN:=(NOT(SOL_TH) AND NOT(LS_THBack)) OR ((SOL_TH) AND LS_THBack), PT:=t#2s);
	IF TON1[0].Q THEN
	Error_LS_THBack:=TRUE;
	END_IF;
	(*節流出磁簧開關*)
	TON1[1](IN:=((SOL_TH) AND NOT(LS_THOut)) OR (NOT(SOL_TH) AND LS_THOut), PT:=t#2s);
	IF TON1[1].Q THEN
	Error_LS_THOut:=TRUE;
	END_IF;
	
	(*前後歸磁簧開關*)
	TON1[2](IN:=(NOT(SOL_Move) AND NOT(LS_MoveBack)) OR ((SOL_Move) AND LS_MoveBack), PT:=t#4s);
	IF TON1[2].Q THEN
	Error_LS_MoveBack:=TRUE;
	END_IF;
	(*前後出磁簧開關*)
	TON1[3](IN:=((SOL_Move) AND NOT(LS_MoveOut)) OR (NOT(SOL_Move) AND LS_MoveOut), PT:=t#4s);
	IF TON1[3].Q THEN
	Error_LS_MoveOut:=TRUE;
	END_IF;
	
	(*夾爪歸磁簧開關*)
	TON1[4](IN:=(NOT(SOL_Clip) AND NOT(LS_ClipBack)) OR ((SOL_Clip) AND LS_ClipBack), PT:=t#2s);
	IF TON1[4].Q THEN
	Error_LS_ClipBack:=TRUE;
	END_IF;
	(*夾爪出磁簧開關*)
	TON1[5](IN:=((SOL_Clip) AND NOT(LS_ClipOut)) OR (NOT(SOL_Clip) AND LS_ClipOut), PT:=t#2s);
	IF TON1[5].Q THEN
	Error_LS_ClipOut:=TRUE;
	END_IF;
END_IF;

//ESTOP
TON1[6](IN:=P_On,PT:=t#1s);
IF NOT(EStopPB) AND TON1[6].Q THEN
	Error_EStopPB:=TRUE;
END_IF;
//SERVO
IF MC_Axis000.DrvStatus.DrvAlarm AND TON1[6].Q THEN
	Error_Servo_UpDown:=TRUE;
END_IF;
IF MC_Axis001.DrvStatus.DrvAlarm AND TON1[6].Q THEN
	Error_Servo_Move:=TRUE;
END_IF;

//定位
IF AutoStatus AND TON1[6].Q AND SystemReadyStatus AND NOT(SNR_MCInPosition) THEN
	Error_SNR_MCInPosition:=TRUE;
END_IF;

(*異常*)
ErrorStatus:=
Error_LS_MoveBack OR
Error_LS_MoveOut OR
Error_LS_ClipBack OR
Error_LS_ClipOut OR
Error_EStopPB OR
Error_Servo_UpDown OR
Error_Servo_Move OR 
Error_SNR_MCInPosition;

ErrorStatusTH:=
Error_LS_THBack OR
Error_LS_THOut;

(*復歸*)
IF PB_Reset THEN
	Error_LS_THBack:=FALSE;
	Error_LS_THOut:=FALSE;
	Error_LS_MoveBack:=FALSE;
	Error_LS_MoveOut:=FALSE;
	Error_LS_ClipBack:=FALSE;
	Error_LS_ClipOut:=FALSE;
	Error_EStopPB:=FALSE;
	Error_Servo_UpDown:=FALSE;
	Error_Servo_Move:=FALSE;
	Error_SNR_MCInPosition:=FALSE;
END_IF;
END_PROGRAM

PROGRAM prConverter
VAR_EXTERNAL
    SV_ServoMoveJogSpeed : LREAL;
    SV_ServoMoveJogSpeed_R : REAL;
    SV_ServoUpdownJogSpeed : LREAL;
    SV_ServoUpdownJogSpeed_R : REAL;
    SV_MoveAbsSpeed : LREAL;
    SV_MoveAbsSpeed_R : REAL;
    SV_UpDownAbsSpeed : LREAL;
    SV_UpDownAbsSpeed_R : REAL;
    State_Homed_Move : BOOL;
END_VAR
VAR_EXTERNAL CONSTANT
    MC_Axis000 : _sAXIS_REF;
    MC_Axis001 : _sAXIS_REF;
END_VAR
VAR_EXTERNAL
    State_Homed_Updown : BOOL;
    State_HomeSerching_Move : BOOL;
    AxMove : stAxis;
    State_HomeSerching_Updown : BOOL;
    AxUpDown : stAxis;
    State_Homed_MC : BOOL;
    State_Homing_MC : BOOL;
    FullNotExistTime : LINT;
    FullNotExistTime_INT : INT;
    FullExistTime_INT : INT;
    FullExistTime : LINT;
    FullNotExistErrorTime : LINT;
    FullNotExistErrorTime_INT : INT;
    FeedExistTime : LINT;
    FeedExistTime_INT : INT;
    FeedNotExistTime : LINT;
    FeedNotExistTime_INT : INT;
END_VAR
SV_ServoMoveJogSpeed:=REAL_TO_LREAL(SV_ServoMoveJogSpeed_R);
SV_ServoUpdownJogSpeed:=REAL_TO_LREAL(SV_ServoUpdownJogSpeed_R);
SV_MoveAbsSpeed:=REAL_TO_LREAL(SV_MoveAbsSpeed_R);
SV_UpDownAbsSpeed:=REAL_TO_LREAL(SV_UpDownAbsSpeed_R);
State_Homed_Move:=MC_Axis001.Details.Homed;
State_Homed_Updown:=MC_Axis000.Details.Homed;
State_HomeSerching_Move:=AxMove.bHoming;
State_HomeSerching_Updown:=AxUpDown.bHoming;
State_Homed_MC:=State_Homed_Move AND State_Homed_Updown AND NOT(State_Homing_MC);
State_Homing_MC:=State_HomeSerching_Move OR State_HomeSerching_Updown;
FullNotExistTime:=INT_TO_LINT(FullNotExistTime_INT);
FullExistTime:=INT_TO_LINT(FullExistTime_INT);
FullNotExistErrorTime:=INT_TO_LINT(FullNotExistErrorTime_INT);
FeedNotExistTime:=INT_TO_LINT(FeedNotExistTime_INT);
FeedExistTime:=INT_TO_LINT(FeedExistTime_INT);
END_PROGRAM

FUNCTION_BLOCK Full
VAR
    AutoFlow : INT;
    TON_Auto1 : TON;
    TON_Auto2 : TON;
    TON_Auto3 : TON;
    tItemNotExistDelayTime : TIME;
    tItemExistTime : TIME;
    tItemNotExistErrorTime : TIME;
END_VAR
VAR_INPUT
    bFullSNR : BOOL;
    iItemNotExistDelayTime : LINT;
    iItemExistTime : LINT;
    iItemNotExistErrorTime : LINT;
END_VAR
VAR_OUTPUT
    bFullRY : BOOL;
    bFullSNRError : BOOL;
END_VAR
VAR_EXTERNAL
    SystemReadyStatus : BOOL;
END_VAR
(******************************************************************
程式:振動筒程序
作者:蔡相偉
版本資訊:v1.0		2016/4/16
******************************************************************)
//時間轉換
tItemNotExistDelayTime:=NanoSecToTime(In:=iItemNotExistDelayTime*100000000);
tItemExistTime:=NanoSecToTime(In:=iItemExistTime*100000000);
tItemNotExistErrorTime:=NanoSecToTime(In:=iItemNotExistErrorTime*100000000);
(*流程*)
(*PowerOn=0*)
IF NOT(SystemReadyStatus) THEN
	AutoFlow:=0;
END_IF;

(*Idle=1*)
IF AutoFlow=0 AND SystemReadyStatus THEN
	AutoFlow:=1;
END_IF;

IF AutoFlow=3 THEN
	AutoFlow:=1;
END_IF;

(*振動筒起振=2*)
TON_Auto1(IN:=AutoFlow=1 AND NOT(bFullSNR) , PT:=tItemNotExistDelayTime);
IF AutoFlow=1 AND TON_Auto1.Q THEN
	AutoFlow:=2;
END_IF;

(*振動筒停振=3*)
TON_Auto2(IN:=AutoFlow=2 AND bFullSNR , PT:=tItemExistTime);
TON_Auto3(IN:=NOT(bFullSNR) AND bFullRY, PT:=tItemNotExistErrorTime);
IF AutoFlow=2 AND TON_Auto2.Q THEN
	AutoFlow:=3;
END_IF;
(******************************************************************)
(*輸出*)
(*振動筒繼電器*)
IF AutoFlow=2 THEN
	bFullRY:=TRUE;
	ELSE
	bFullRY:=FALSE;
END_IF;
(*振動筒滿料異常*)
IF AutoFlow=2 AND (TON_Auto3.Q) THEN
	bFullSNRError:=TRUE;
	ELSE
	bFullSNRError:=FALSE;
END_IF;
END_FUNCTION_BLOCK

FUNCTION_BLOCK fbFeed
VAR
    tNoObjDelayTime : TIME;
    tObjectExistDelayTime : TIME;
    Autoflow : INT;
    TON_1 : TON;
    TON_2 : TON;
    TON_3 : TON;
    ObjSNRStatus : BOOL;
    THStatus : BOOL;
    R_TRIG_1 : R_TRIG;
    R_TRIG_2 : R_TRIG;
    R_TRIG_3 : R_TRIG;
    R_TRIG_4 : R_TRIG;
END_VAR
VAR_INPUT
    wNoObjDelayTime : LINT;
    wObjectExistDelayTime : LINT;
    bReset : BOOL;
    bTHPB : BOOL;
    bObjSNR : BOOL;
    bFeedStart : BOOL;
    bTHBackLS : BOOL;
    bTHOutLS : BOOL;
    bErrorTHBack : BOOL;
    bErrorTHOut : BOOL;
    bInterlock_thback : BOOL;
    bInterlock_thout : BOOL;
    bSupplierRY : BOOL;
END_VAR
VAR_OUTPUT
    bFeedError : BOOL;
    bFeedFinish : BOOL;
    bTHSOL : BOOL;
    bFeedRY : BOOL;
END_VAR
VAR_EXTERNAL
    SystemReadyStatus : BOOL;
    AutoStatus : BOOL;
END_VAR
(*************************************************************************
程序名稱:平送FB
作者:蔡相偉
版本,日期,版本資訊:
1.0.0	2016/6/28		初始版本

PowerOn=0
Idle=1
無料,節流出=2
到出,平送起振=3
工件到位,平送停振=4
節流回=5
節流到回=6
*************************************************************************)
//時間轉換
tNoObjDelayTime:=NanoSecToTime(wNoObjDelayTime*100000000);
tObjectExistDelayTime:=NanoSecToTime(wObjectExistDelayTime*100000000);

//PowerOn=0
IF Autoflow=0 AND SystemReadyStatus AND NOT(bErrorTHBack) AND NOT(bErrorTHOut) AND AutoStatus  THEN
	Autoflow:=1;
END_IF;

(*Idle=1*)
TON_1(IN:= Autoflow=1 AND NOT(bObjSNR) ,PT:= tNoObjDelayTime);
IF Autoflow=1 AND (bFeedStart) THEN
	Autoflow:=2;
END_IF;
(*無料,節流出=2*)
IF Autoflow=2 THEN
	ObjSNRStatus:=FALSE;
END_IF;

IF Autoflow=2 AND bTHOutLS THEN
	Autoflow:=3;
END_IF;
(*到出,平送起振=3*)
IF Autoflow=3 AND bObjSNR THEN
	ObjSNRStatus:=TRUE;
END_IF;
TON_2(IN:= Autoflow=3 AND ObjSNRStatus ,PT:= tObjectExistDelayTime);
TON_3(IN:= Autoflow=3 AND NOT(ObjSNRStatus) ,PT:= t#4s);
IF TON_3.Q THEN
	bFeedError:=TRUE;
END_IF;
IF bReset THEN
	bFeedError:=FALSE;
END_IF;

IF Autoflow=3 AND TON_2.Q AND NOT(bFeedError) THEN
	Autoflow:=4;
END_IF;
(*工件到位,平送停振=4*)
IF Autoflow=4 THEN
	Autoflow:=5;
END_IF;
(*節流回=5*)
IF Autoflow=5 AND bTHBackLS THEN
	Autoflow:=6;
END_IF;
(*節流到回=6*)
IF Autoflow=6 THEN
	bFeedFinish:=TRUE;
	ELSE
	bFeedFinish:=FALSE;
END_IF;

IF Autoflow=6 AND NOT(bFeedStart) THEN
	Autoflow:=1;
END_IF;
(*************************************************************************)
(*Error*)
R_TRIG_3(CLK:=bErrorTHBack);
R_TRIG_4(CLK:=bErrorTHOut);

IF NOT(SystemReadyStatus) OR NOT(AutoStatus) OR bErrorTHBack OR bErrorTHOut THEN
	Autoflow:=0;
END_IF;

(*************************************************************************)
(*手動*)
(*節流*)
R_TRIG_1(CLK:=bTHPB AND NOT(AutoStatus));
(*SET*)
IF (((R_TRIG_1.Q) AND NOT(THStatus)) OR Autoflow=2 OR R_TRIG_3.Q) AND bInterlock_thout THEN
	bTHSOL:=TRUE;
END_IF;
(*RESET*)
IF (((R_TRIG_1.Q) AND THStatus) OR Autoflow=5 OR R_TRIG_4.Q) AND bInterlock_thback THEN
	bTHSOL:=FALSE;
END_IF;
(*STATE*)
THStatus:=bTHSOL;

(*平送*)
(*輸出*)
bFeedRY:=Autoflow=2 OR Autoflow=3 OR bSupplierRY OR bTHSOL;
END_FUNCTION_BLOCK